Omron CX-Programmer project NuevoProyecto (CX-Programmer 9.61)

# PLC NuevoPLC1: CQM1 CPU41

## Program NuevoPrograma1 (no task)
Local symbols
CMP 255.06 BOOL
CNT BOOL
EM 117.10 BOOL
Etapa 116.02 BOOL
Etapa0 116.00 BOOL
Etapa1 116.01 BOOL
Etapa10 116.10 BOOL
Etapa11 116.11 BOOL
Etapa12 116.12 BOOL
Etapa13 116.13 BOOL
Etapa14 116.14 BOOL
Etapa15 116.15 BOOL
Etapa16 117.00 BOOL
Etapa17 117.02 BOOL
Etapa19 117.03 BOOL
Etapa2 116.02 BOOL
Etapa20 117.05 BOOL
Etapa21 117.06 BOOL
Etapa22 117.07 BOOL
Etapa23 117.08 BOOL
Etapa24 117.09 BOOL
Etapa25 117.11 BOOL
Etapa26 BOOL
Etapa27 117.12 BOOL
Etapa3 116.03 BOOL
Etapa30 117.13 BOOL
Etapa31 117.14 BOOL
Etapa4 116.04 BOOL
Etapa5 116.05 BOOL
Etapa6 116.06 BOOL
Etapa7 116.07 BOOL
Etapa8 116.08 BOOL
Etapa9 116.09 BOOL
FCB 0.04 BOOL
FCD 0.05 BOOL
FCE 0.07 BOOL
FCI 0.08 BOOL
FCN 0.06 BOOL
FCS 0.00 BOOL
FM1 0.10 BOOL
FM2 0.09 BOOL
FcI BOOL
HM1 100.07 BOOL
HM2 100.01 BOOL
HRO UINT_BCD
KMDM2 100.00 BOOL
KMI 100.02 BOOL  ; Contactor marcha izquierda
KMI1 100.02 BOOL  ; Contactor marcha izquierda
KMIM1 100.05 BOOL
LA 100.13 BOOL  ; Lámpara de avería
LACTM1 100.07 BOOL
LACTM2 100.01 BOOL
LAVM1 100.15 BOOL
LAVM2 100.13 BOOL
LF 100.14 BOOL  ; Lámpara de funcionamiento
M1 0.12 BOOL
M1DER 100.05 BOOL  ; Contactor marcha derecha
M1Der 100.06 BOOL
M1EM 100.15 BOOL
M1IZQ 100.06 BOOL
M1Izq 100.05 BOOL
M1_AUX_DER BOOL
M1_DER_AUX 20.04 BOOL
M1_IZQ_AUX 20.03 BOOL
M2 0.13 BOOL
M2B 100.08 BOOL
M2BAJAR 100.08 BOOL
M2EM 100.13 BOOL
M2S 100.00 BOOL
M2SUBIR 100.00 BOOL  ; Contactor marcha derecha
M2_BAJAR_AUX 20.02 BOOL
M2_SUBIR_AUX 20.01 BOOL
PM 0.14 BOOL
PMD 0.05 BOOL  ; Pulsador marcha derecha
PMDM1 200.02 BOOL
PMDM2 200.03 BOOL
PMI 0.02 BOOL  ; Pulsador de marcha izquierda
PMIM1 200.01 BOOL
PMIM2 200.04 BOOL
PP 0.15 BOOL
P_0N BOOL
P_ON BOOL
RT 0.13 BOOL  ; Contacto relé térmico
SensorTemperatura 0.11 BOOL
eTAPA21 BOOL

### Section Sección1

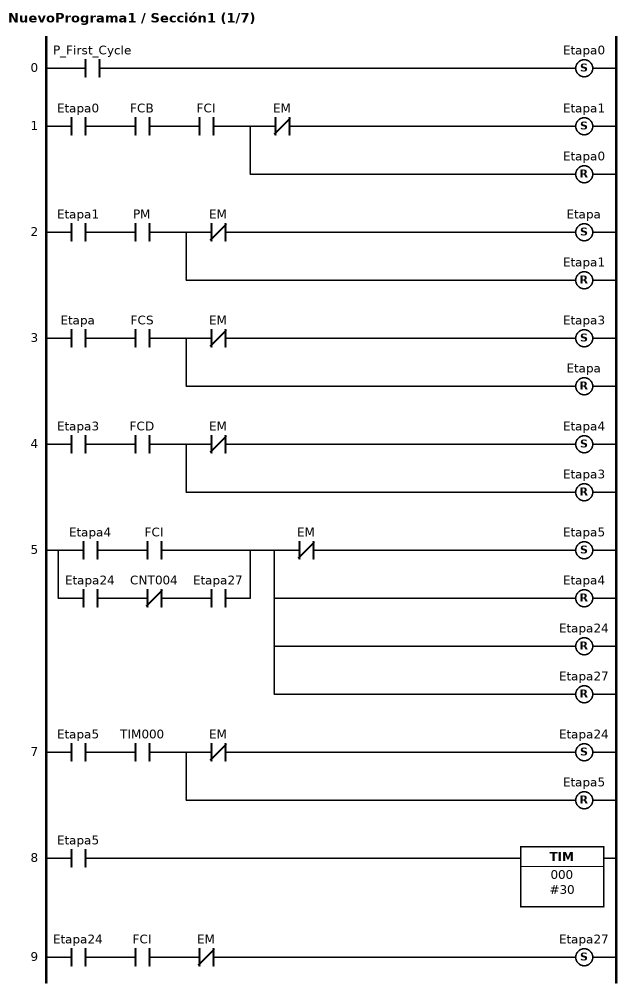
; rung 0
LD P_First_Cycle
SET Etapa0
; rung 1
LD Etapa0
AND FCB
AND FCI
OUT TR0
ANDNOT EM
SET Etapa1
LD TR0
RSET Etapa0
; rung 2
LD Etapa1
AND PM
OUT TR0
ANDNOT EM
SET Etapa
LD TR0
RSET Etapa1
; rung 3
LD Etapa
AND FCS
OUT TR0
ANDNOT EM
SET Etapa3
LD TR0
RSET Etapa
; rung 4
LD Etapa3
AND FCD
OUT TR0
ANDNOT EM
SET Etapa4
LD TR0
RSET Etapa3
; rung 5
LD Etapa4
AND FCI
LD Etapa24
ANDNOT CNT004
AND Etapa27
ORLD
OUT TR0
ANDNOT EM
SET Etapa5
LD TR0
RSET Etapa4
RSET Etapa24
RSET Etapa27
; rung 7
LD Etapa5
AND TIM000
OUT TR0
ANDNOT EM
SET Etapa24
LD TR0
RSET Etapa5
; rung 8
LD Etapa5
TIM 000 #30
; rung 9
LD Etapa24
AND FCI
ANDNOT EM
SET Etapa27

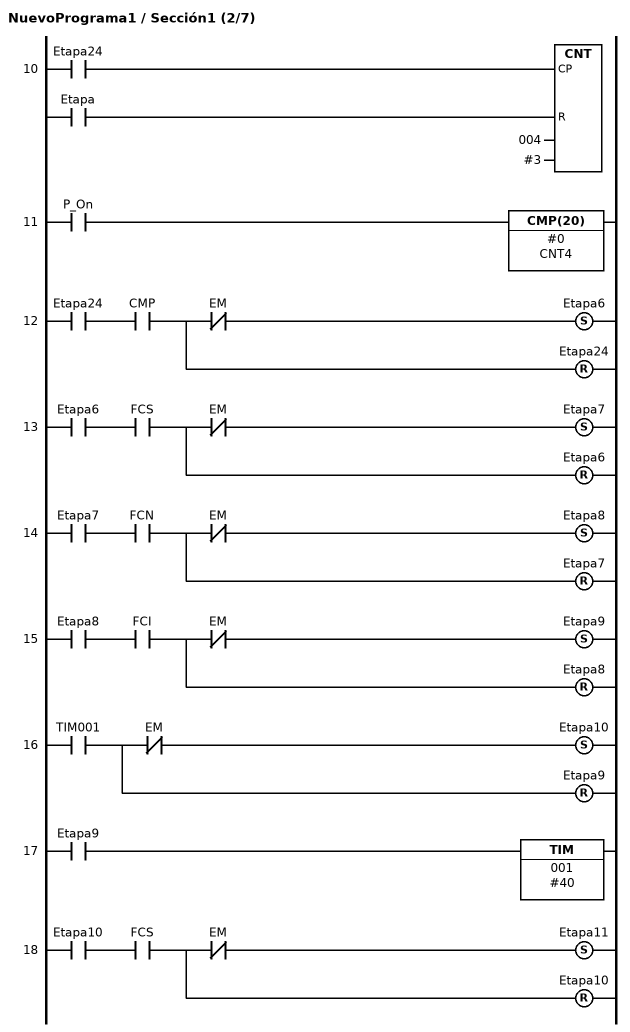
; rung 10
LD Etapa24
LD Etapa
CNT 004 #3
; rung 11
LD P_On
CMP(20) #0 CNT4
; rung 12
LD Etapa24
AND CMP
OUT TR0
ANDNOT EM
SET Etapa6
LD TR0
RSET Etapa24
; rung 13
LD Etapa6
AND FCS
OUT TR0
ANDNOT EM
SET Etapa7
LD TR0
RSET Etapa6
; rung 14
LD Etapa7
AND FCN
OUT TR0
ANDNOT EM
SET Etapa8
LD TR0
RSET Etapa7
; rung 15
LD Etapa8
AND FCI
OUT TR0
ANDNOT EM
SET Etapa9
LD TR0
RSET Etapa8
; rung 16
LD TIM001
OUT TR0
ANDNOT EM
SET Etapa10
LD TR0
RSET Etapa9
; rung 17
LD Etapa9
TIM 001 #40
; rung 18
LD Etapa10
AND FCS
OUT TR0
ANDNOT EM
SET Etapa11
LD TR0
RSET Etapa10

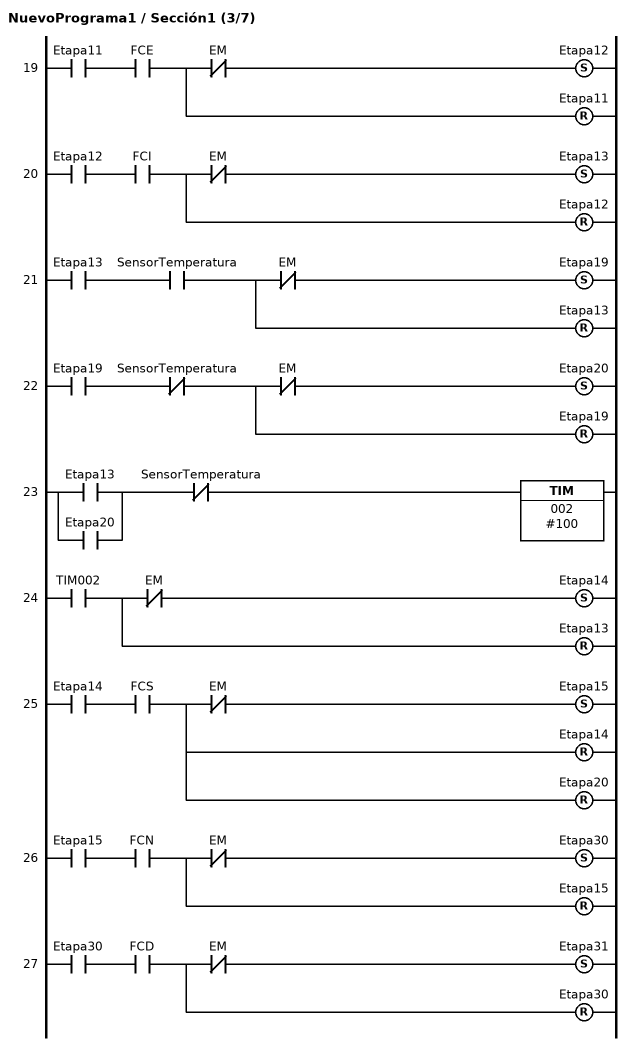
; rung 19
LD Etapa11
AND FCE
OUT TR0
ANDNOT EM
SET Etapa12
LD TR0
RSET Etapa11
; rung 20
LD Etapa12
AND FCI
OUT TR0
ANDNOT EM
SET Etapa13
LD TR0
RSET Etapa12
; rung 21
LD Etapa13
AND SensorTemperatura
OUT TR0
ANDNOT EM
SET Etapa19
LD TR0
RSET Etapa13
; rung 22
LD Etapa19
ANDNOT SensorTemperatura
OUT TR0
ANDNOT EM
SET Etapa20
LD TR0
RSET Etapa19
; rung 23
LD Etapa13
OR Etapa20
ANDNOT SensorTemperatura
TIM 002 #100
; rung 24
LD TIM002
OUT TR0
ANDNOT EM
SET Etapa14
LD TR0
RSET Etapa13
; rung 25
LD Etapa14
AND FCS
OUT TR0
ANDNOT EM
SET Etapa15
LD TR0
RSET Etapa14
RSET Etapa20
; rung 26
LD Etapa15
AND FCN
OUT TR0
ANDNOT EM
SET Etapa30
LD TR0
RSET Etapa15
; rung 27
LD Etapa30
AND FCD
OUT TR0
ANDNOT EM
SET Etapa31
LD TR0
RSET Etapa30

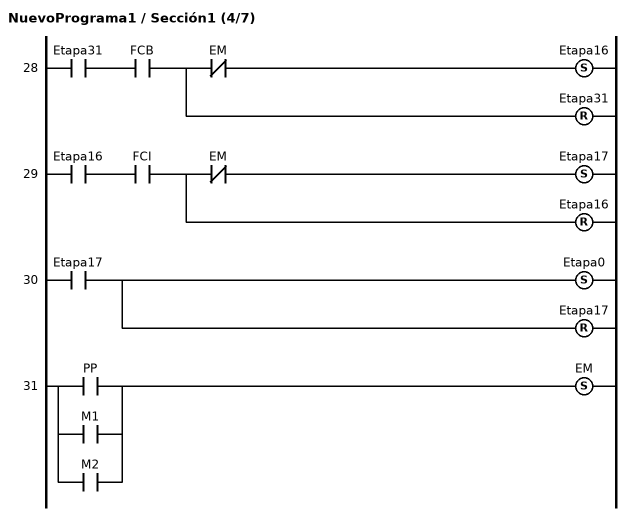
; rung 28
LD Etapa31
AND FCB
OUT TR0
ANDNOT EM
SET Etapa16
LD TR0
RSET Etapa31
; rung 29
LD Etapa16
AND FCI
OUT TR0
ANDNOT EM
SET Etapa17
LD TR0
RSET Etapa16
; rung 30
LD Etapa17
SET Etapa0
RSET Etapa17
; rung 31
LD PP
OR M1
OR M2
SET EM

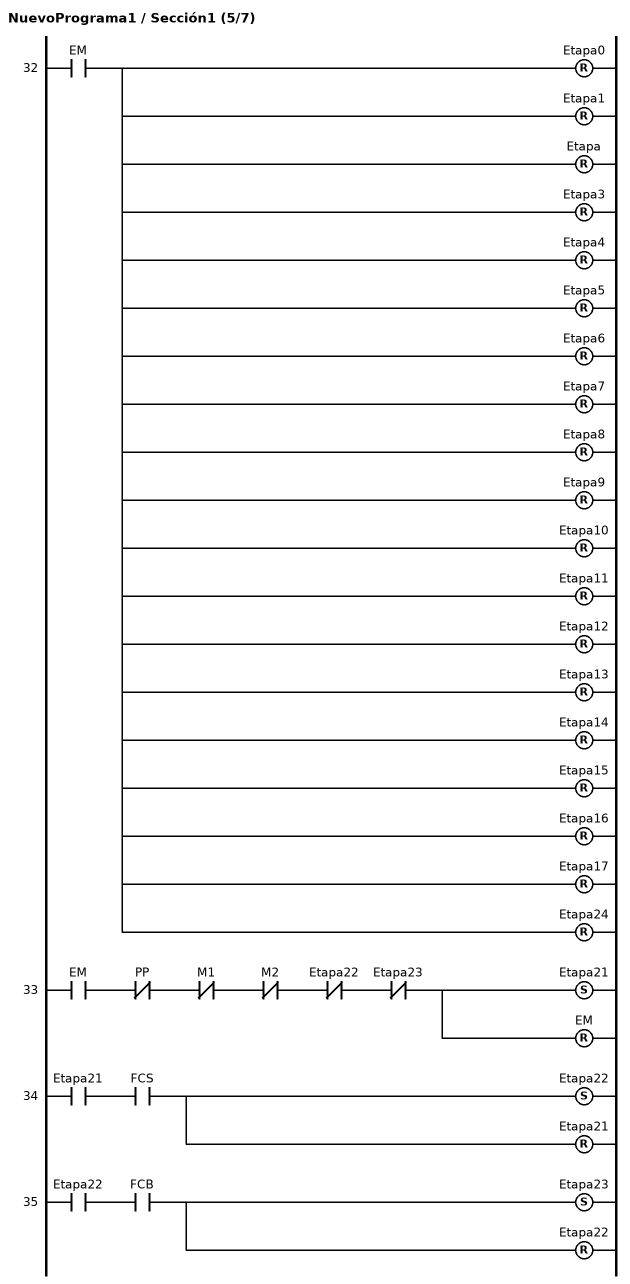
; rung 32
LD EM
RSET Etapa0
RSET Etapa1
RSET Etapa
RSET Etapa3
RSET Etapa4
RSET Etapa5
RSET Etapa6
RSET Etapa7
RSET Etapa8
RSET Etapa9
RSET Etapa10
RSET Etapa11
RSET Etapa12
RSET Etapa13
RSET Etapa14
RSET Etapa15
RSET Etapa16
RSET Etapa17
RSET Etapa24
; rung 33
LD EM
ANDNOT PP
ANDNOT M1
ANDNOT M2
ANDNOT Etapa22
ANDNOT Etapa23
SET Etapa21
RSET EM
; rung 34
LD Etapa21
AND FCS
SET Etapa22
RSET Etapa21
; rung 35
LD Etapa22
AND FCB
SET Etapa23
RSET Etapa22

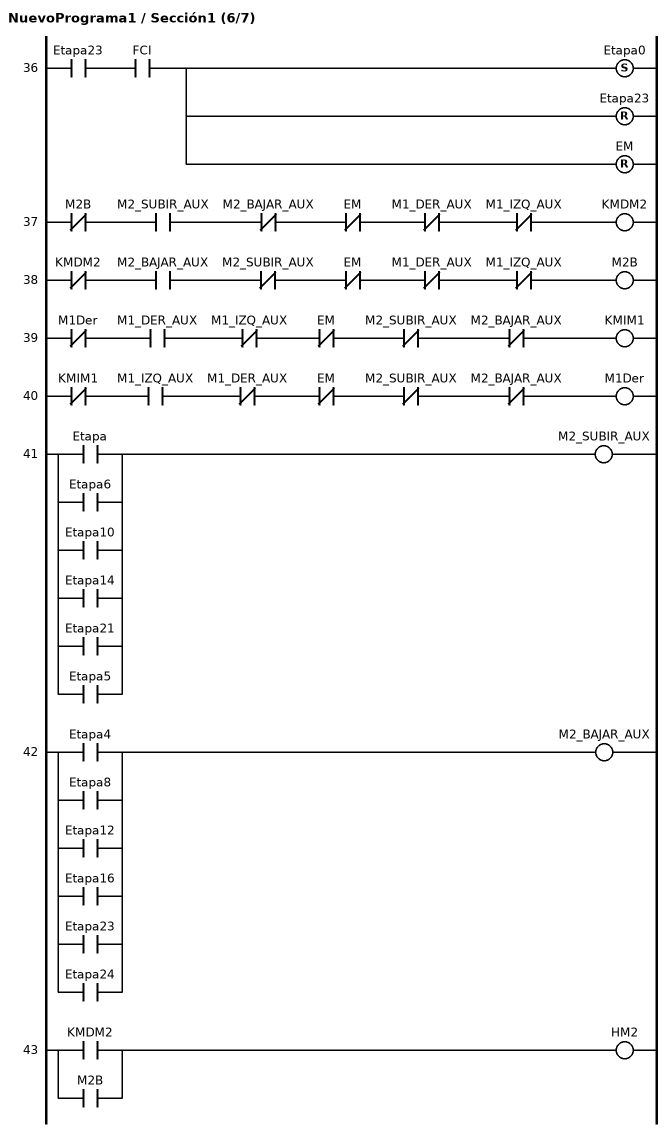
; rung 36
LD Etapa23
AND FCI
SET Etapa0
RSET Etapa23
RSET EM
; rung 37
LDNOT M2B
AND M2_SUBIR_AUX
ANDNOT M2_BAJAR_AUX
ANDNOT EM
ANDNOT M1_DER_AUX
ANDNOT M1_IZQ_AUX
OUT KMDM2
; rung 38
LDNOT KMDM2
AND M2_BAJAR_AUX
ANDNOT M2_SUBIR_AUX
ANDNOT EM
ANDNOT M1_DER_AUX
ANDNOT M1_IZQ_AUX
OUT M2B
; rung 39
LDNOT M1Der
AND M1_DER_AUX
ANDNOT M1_IZQ_AUX
ANDNOT EM
ANDNOT M2_SUBIR_AUX
ANDNOT M2_BAJAR_AUX
OUT KMIM1
; rung 40
LDNOT KMIM1
AND M1_IZQ_AUX
ANDNOT M1_DER_AUX
ANDNOT EM
ANDNOT M2_SUBIR_AUX
ANDNOT M2_BAJAR_AUX
OUT M1Der
; rung 41
LD Etapa
OR Etapa6
OR Etapa10
OR Etapa14
OR Etapa21
OR Etapa5
OUT M2_SUBIR_AUX
; rung 42
LD Etapa4
OR Etapa8
OR Etapa12
OR Etapa16
OR Etapa23
OR Etapa24
OUT M2_BAJAR_AUX
; rung 43
LD KMDM2
OR M2B
OUT HM2

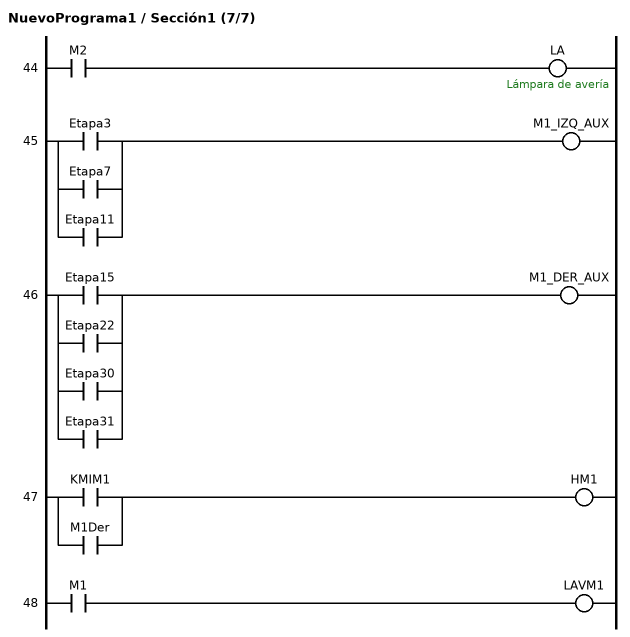
; rung 44
LD M2
OUT LA  ; Lámpara de avería
; rung 45
LD Etapa3
OR Etapa7
OR Etapa11
OUT M1_IZQ_AUX
; rung 46
LD Etapa15
OR Etapa22
OR Etapa30
OR Etapa31
OUT M1_DER_AUX
; rung 47
LD KMIM1
OR M1Der
OUT HM1
; rung 48
LD M1
OUT LAVM1

### Section END
; rung 0
END(01)